TYPE k_Daten :
STRUCT
	k_Kalibrierung : ARRAY [1..4,1..5] OF REAL; // Array [WaagenNummer, Kalibrierungsschritt]
END_STRUCT
END_TYPE

(* stored: Version 1.1.0.1, ProductVersion 3.1.4019.2
   DUT k_Daten: Id {fab6a44b-731e-4818-bb13-99b5c8e7a2dd} *)
